(*	Sample Code Disclaimer
	All sample code provided by Beckhoff Automation LLC are for illustrative purposes only
	and are provided “as is” and without any warranties, express or implied.
	Actual implementations in applications will vary significantly.
	Beckhoff Automation LLC shall have no liability for, and does not waive any rights in relation to,
	any code samples that it provides or the use of such code samples for any purpose.
*)
FUNCTION_BLOCK FB_Drive_AX5000 EXTENDS FB_ComponentBase IMPLEMENTS I_Drive_AX5000
VAR
	// Properties
	_SercosErrorID: UINT;
	// References
	refAxis: REFERENCE TO AXIS_REF;
	
	// Method Requests
	DriveResetReq: BOOL;
	
	// General
	fbSoEReset: FB_SoEReset;
	
	
	
	{attribute 'hide'}
	DummyAxis	  : AXIS_REF;
	_ErrorSercoID: INT;
END_VAR

METHOD CyclicLogic : BOOL
VAR_INPUT
END_VAR

VAR
	_ErrorSercoID: UINT;
END_VAR
// Call Super
SUPER^.CyclicLogic();

// Drive Reset Request
IF DriveResetReq THEN
	fbSoEReset.Execute := TRUE;
	DriveResetReq := FALSE;
ELSE
	fbSoEReset.Execute := FALSE;
END_IF

// Call AX5000 SERCOS Reset
fbSoEReset(Axis:= refAxis);

// Busy Logic
IF NOT fbSoEReset.Busy THEN
	_Busy := FALSE;
END_IF

// Error Logic
IF fbSoEReset.Error THEN
	_Busy := FALSE;
	_Error := TRUE;
	_ErrorID := fbSoEReset.AdsErrId;
	_SercosErrorID := fbSoEReset.SercosErrId;
END_IF
END_METHOD

METHOD DriveReset : BOOL
// Call Super
SUPER^.Reset();

IF NOT __ISVALIDREF(refAxis) OR _Busy THEN
    RETURN;
END_IF

_Busy        := TRUE;
_Error       := FALSE;
_ErrorID     := 0;
_SercosErrorID := 0;
DriveResetReq := TRUE;

DriveReset := TRUE;
END_METHOD

//! @summary Basic component initialization logic
METHOD PROTECTED Initialize : BOOL;

//! @description This method is called by <c>CyclicLogic()</c> as required
refAxis REF= DummyAxis;

fbSoEReset.Execute := FALSE;

Initialize := SUPER^.Initialize();
END_METHOD

{warning 'add property implementation'}
PROPERTY REF_Axis : REFERENCE TO AXIS_REF
GET
REF_Axis REF= refAxis;
END_GET
SET
refAxis REF= REF_Axis;
END_SET
END_PROPERTY

{warning 'add property implementation'}
PROPERTY SercosErrorID : UINT
GET
SercosErrorID := _SercosErrorID;
END_GET
END_PROPERTY

END_FUNCTION_BLOCK

(* stored: Version 1.1.0.1, ProductVersion 3.1.4024.12
   POU FB_Drive_AX5000: Id {753d2ad4-0317-4039-aaaf-2342ef9391ce}, SpecialFunc None
   Folder BaseComponent: Id {e6390556-2426-4c18-8267-15aa8a2a601c}
   Method CyclicLogic: Id {c06a9a03-f364-4b21-96d1-4959359d2b5a}
   Method DriveReset: Id {d5c0017f-0242-4a80-9944-b64b963b97c3}
   Method Initialize: Id {45f5b00b-210f-4397-bbaa-379d19c5f3ce}
   Property REF_Axis: Id {18b34b49-6146-4624-8860-1c2da4f36b41}
   Get Get: Id {998e4c27-d3bb-4835-ba5d-43d681e13047}
   Set Set: Id {3d5a81e5-9fce-46b5-8b62-4501391fc32d}
   Property SercosErrorID: Id {d9861e40-539f-4899-95f4-fcea5cc4fdc9}
   Get Get: Id {3c839203-23b7-422a-806e-6c1eb118b39d} *)
